# EPICS autosave request: tomoStreamApp/Db/tomoStream_settings.req
# This file is used by autosave to determine what PVs to save
# It is also used by tomoStream to determine what PVs to create

# This file contains all of the PVs used by the tomostream base class.

# Lines that begin with #controlPV are not saved by autosave,
# but they are used by tomostream.
# These PVs are not saved in the tomostream configuration file.

############################
# Streaming analysis control
############################
$(P)$(R)StreamStatus
$(P)$(R)StreamBufferSize
$(P)$(R)StreamCenter
$(P)$(R)StreamFilterType
$(P)$(R)StreamOrthoX
$(P)$(R)StreamOrthoY
$(P)$(R)StreamOrthoZ
$(P)$(R)StreamReconTime
